// TwinCAT 3 PLC project PLC
// ProgramVersion: 3.1.4023.0
// libraries:
//   Tc2_Standard, * (Beckhoff Automation GmbH)
//   Tc2_System, * (Beckhoff Automation GmbH)
//   Tc2_Utilities, * (Beckhoff Automation GmbH)
//   Tc3_IotBase, * (Beckhoff Automation GmbH)
//   Tc3_Module, * (Beckhoff Automation GmbH)
// project tree:
//   / PlcTask.TcTTO
//   POUs/ FBGenerateData.TcPOU, MAIN.TcPOU, ST_SensorData.TcDUT, To_InfluxDb.TcPOU
// real-time tasks:
//   TASK PlcTask: cycle T#10ms, priority 20, ADS port 350

CONFIGURATION PLC
    RESOURCE PLC ON TwinCAT3
        TASK PlcTask(INTERVAL := T#10ms, PRIORITY := 20);
        PROGRAM MAIN WITH PlcTask : MAIN;
    END_RESOURCE
END_CONFIGURATION

// ---- POUs/ST_SensorData.TcDUT
TYPE ST_SensorData :
STRUCT
	sSensorId : STRING:='';
	rSensorValue : REAL;
END_STRUCT
END_TYPE

// ---- POUs/MAIN.TcPOU
PROGRAM MAIN
VAR
	Influx : To_InfluxDb;
	bExecute: BOOL;
	tTime: TIME := T#1s;
	bBusy: BOOL;
	bError: BOOL;
	bErrorId: DINT;
	stSensors : ARRAY[0..10] OF ST_SensorData;
	Generatedata : FBGenerateData;
	tIntervalTimer: TON;
	sHostName: STRING;
END_VAR

stSensors[0].sSensorId := '1PT01';
Generatedata(data:=stSensors[0]);
stSensors[1].sSensorId := '1PT02';
Generatedata(data:=stSensors[1]);
stSensors[2].sSensorId := '1PT03';
Generatedata(data:=stSensors[2]);
stSensors[3].sSensorId := '1PT04';
Generatedata(data:=stSensors[3]);
stSensors[4].sSensorId := '1PT05';
Generatedata(data:=stSensors[4]);
stSensors[5].sSensorId := '1PT06';
Generatedata(data:=stSensors[5]);


// Send data to InfluxDb
Influx(
	bExecute:= bExecute, 
	tInterval:= tTime, 
	sHostName:= '127.0.0.1', 
	nHostPort:= 8086, 
	sDatabaseName:= 'SensorData',
	sMeasurementName:= 'PtData',
	stData:= stSensors, 
	bBusy=> bBusy, 
	bError=> bError, 
	nErrId=> bErrorId);

END_PROGRAM

// ---- POUs/To_InfluxDb.TcPOU
FUNCTION_BLOCK To_InfluxDb

VAR_INPUT
	bExecute: BOOL;		// Start logging when high. 
	tInterval: TIME;	// How often to log.
	sHostName: STRING;	// Ip-adress to Db
	nHostPort: UINT; // Influxdb is at 8086 default 
	sDatabaseName: STRING; // Db name
	sMeasurementName: STRING; // "Tablename"
	stData: ARRAY[0..10] OF ST_SensorData; // Data to be logged 
END_VAR
VAR_OUTPUT
	bBusy: BOOL;
	bError: BOOL;
	nErrId: DINT;
END_VAR
VAR
	nIndex: INT;
	nState: INT;
	nErrState: INT;
	sUri: STRING;
	sContent: STRING(32768);
	sData: STRING(255);
	nStartPos: UDINT;
	nLen: UDINT;
	
	tIntervalTimer: TON;
	fbIotHttpClient: FB_IotHttpClient;
	fbIotHttpRequest: FB_IotHttpRequest;
END_VAR

tIntervalTimer(IN:=bExecute AND NOT tIntervalTimer.Q, PT:=tInterval); // Timer for executing the http request.
CASE nState OF
0:	

	IF bExecute THEN
		bBusy:=TRUE;
		bError:=FALSE;
		nState:=10;
	END_IF

10:	

	mInit(); // Initialize HttpClient

20:

	mGenerateBodyContent(); // Generate data string to be sent to InfluxDb
	
21:

	mSendRequest(); // Execute send request
	
22:
	
	mWaitUntilDone(); // Wait until done or error

99:

	mErrorHandling(); // Handle the error if needed.
	
END_CASE

METHOD PRIVATE mErrorHandling : BOOL
bError:=TRUE;
bBusy:=FALSE;
IF NOT bExecute THEN
	nState:=0;
END_IF
END_METHOD

METHOD PRIVATE mGenerateBodyContent : BOOL
IF bExecute THEN
	IF tIntervalTimer.Q THEN
		sUri:=CONCAT('/write?db=', sDatabaseName);
		MEMSET(ADR(sContent),0,SIZEOF(sContent)); // Memset fixed the problems with status 400 and database havoc... 
		nStartPos:=0;
		FOR nIndex:=0 TO 5 DO
			IF stData[nIndex].sSensorId <> '' THEN
				sData:=sMeasurementName; 									nLen:=INT_TO_UDINT(LEN(sData)); MEMMOVE(ADR(sContent)+nStartPos, ADR(sData), nLen); nStartPos:=nStartPos+nLen;
				sData:=',SensorId='; 										nLen:=INT_TO_UDINT(LEN(sData)); MEMMOVE(ADR(sContent)+nStartPos, ADR(sData), nLen); nStartPos:=nStartPos+nLen;
				sData:=stData[nIndex].sSensorId; 							nLen:=INT_TO_UDINT(LEN(sData)); MEMMOVE(ADR(sContent)+nStartPos, ADR(sData), nLen); nStartPos:=nStartPos+nLen;
				sData:=' fSensorValue=';									nLen:=INT_TO_UDINT(LEN(sData)); MEMMOVE(ADR(sContent)+nStartPos, ADR(sData), nLen); nStartPos:=nStartPos+nLen;
				sData:=REAL_TO_STRING(stData[nIndex].rSensorValue);			nLen:=INT_TO_UDINT(LEN(sData)); MEMMOVE(ADR(sContent)+nStartPos, ADR(sData), nLen); nStartPos:=nStartPos+nLen;
				sData:='$n'; 												nLen:=INT_TO_UDINT(LEN(sData)); MEMMOVE(ADR(sContent)+nStartPos, ADR(sData), nLen); nStartPos:=nStartPos+nLen;
			ELSE
				EXIT;
			END_IF
		END_FOR
		nState:=21;
	END_IF	
ELSE
	bBusy:=FALSE;
	nState:=0;
END_IF
END_METHOD

METHOD PRIVATE mInit : BOOL
fbIotHttpClient.sHostName:=sHostName;
fbIotHttpClient.nHostPort:=nHostPort;
fbIotHttpClient.bKeepAlive:=TRUE;
fbIotHttpClient.tConnectionTimeout:=T#10S;
fbIotHttpClient.Execute();
IF fbIotHttpClient.bConfigured THEN
	nState:=20;
ELSIF fbIotHttpClient.bError THEN
	nErrState:=nState;
	nErrId:=fbIotHttpClient.hrErrorCode;
	nState:=99;
END_IF
END_METHOD

METHOD PRIVATE mSendRequest : BOOL

fbIotHttpClient.Execute();	
IF fbIotHttpRequest.SendRequest(
	sUri:=sUri,
	fbClient:=fbIotHttpClient, 
	eRequestType:=ETcIotHttpRequestType.HTTP_POST, 
	pContent:=ADR(sContent), 
	nContentSize:=LEN2(ADR(sContent)), 0)
THEN
	nState:=22;
END_IF
END_METHOD

METHOD PRIVATE mWaitUntilDone : BOOL

fbIotHttpClient.Execute();	
IF fbIotHttpRequest.bError THEN
	nErrState:=nState;
	nErrId:=fbIotHttpRequest.eErrorId;
	nState:=99;
ELSIF NOT fbIotHttpRequest.bBusy THEN
	nState:=20;
END_IF
END_METHOD

END_FUNCTION_BLOCK

// ---- POUs/FBGenerateData.TcPOU
FUNCTION_BLOCK FBGenerateData
VAR_IN_OUT
	data : ST_SensorData;
END_VAR

VAR
	rand : drand;
	value: LREAL;
END_VAR

rand(Seed:=LREAL_TO_INT(value));
value := rand.Num;
data.rSensorValue := LREAL_TO_REAL(value);

END_FUNCTION_BLOCK
